INTERFACE I_DataChannelRecv

PROPERTY Error : INT
SET
END_SET
GET
END_GET
END_PROPERTY

PROPERTY Busy : BOOL
GET
END_GET
END_PROPERTY

{attribute 'object_name' := 'GetData'}
METHOD GetData : BOOL
VAR_INPUT
	udiDataSize: UDINT;
	pData: POINTER TO BYTE;
END_VAR
END_METHOD

{attribute 'object_name' := 'InitChannel'}
METHOD InitChannel : BOOL
VAR_INPUT
	udiDataSize: UDINT;
	pInputData: POINTER TO BYTE;
END_VAR
END_METHOD

PROPERTY DataSize : UDINT
GET
END_GET
END_PROPERTY

END_INTERFACE

(* stored: Version 1.1.0.1, ProductVersion 3.1.0.36
   Itf I_DataChannelRecv: Id {5ca02700-d8cd-48af-917f-71f240b56d30}
   Property Error: Id {0a0c7599-7fc9-411f-839f-d3bb95fc8b43}
   Set Set: Id {928f5267-8917-4501-ae3d-0a309d189145}
   Get Get: Id {983a13a4-7022-4b4a-a144-164ca380b711}
   Property Busy: Id {14e7aced-cca9-4ef1-8ff4-84bef2a36780}
   Get Get: Id {a5beac3c-462d-4878-b3f6-c6a0754d963f}
   Method GetData: Id {d56ae630-d3c3-4371-b896-0fa7b8c9648f}
   Method InitChannel: Id {e51ece68-5c09-424a-927f-f06914d2a6d9}
   Property DataSize: Id {ea5b0838-fffb-4753-9716-b5d8710c2ef7}
   Get Get: Id {1655855d-f069-4fff-a98b-92370e1febea} *)
